Universal Robots PolyScope program: weigh_single_new2.urp

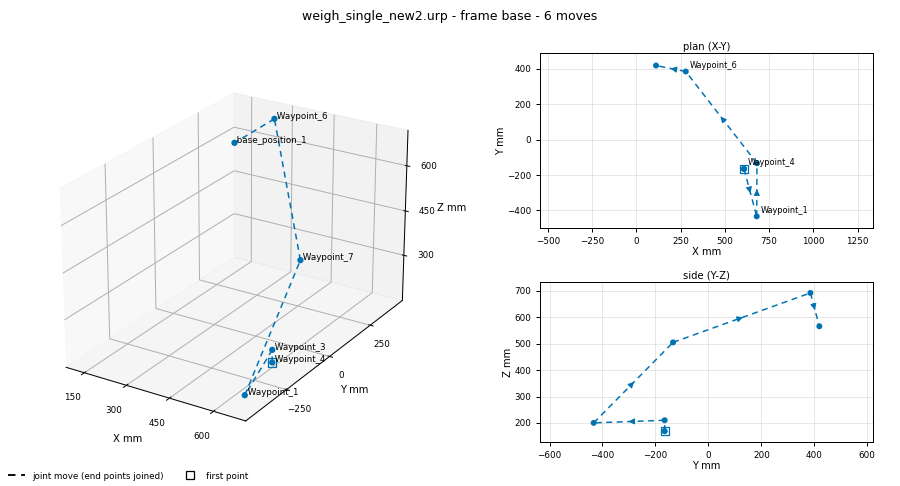
[picture p0: tool path of weigh_single_new2.urp in frame base, 6 of 6 moves have a stored position in this frame; points joined in program order, loops and branches not executed]
Program weigh_single_new2 (installation=default directory=/programs/Nicolas_Arteaga/quality createdIn=5.12.4.1101661 lastSavedIn=5.12.4.1101661 robotSerialNumber=20225502378)
Calibrated DH parameters: a=[0.00022, -0.425328, -0.389701, 0.000059, 0.000065, 0]; d=[0.162608, 0.803456, 9.992211, -10.662202, 0.099702, 0.099559]; alpha=[1.570756, 0.001543, 0.004316, 1.570651, -1.570122, 0]; deltaTheta=[0, 0.002917, 0.116094, -0.119008, 0, -0.000001]
Robot Program (runOnlyOnce=true)
  MoveJ speed 60 deg/s, acceleration 80 deg/s^2 (useActiveTCP=true) feature=Base
    URCap Gripper (Robotiq_Grippers, Robotiq Inc.) dataModel(position=41.96078431372549, force=100.0, speed=100.0, positionInDouble=41.96078431372549, forceInDouble=100.0, speedInDouble=100.0, slaveIds=[9], blocking=true)
    URCap Gripper (Robotiq_Grippers, Robotiq Inc.) dataModel(position=100.0, force=100.0, speed=100.0, positionInDouble=100.0, forceInDouble=100.0, speedInDouble=100.0, slaveIds=[9], blocking=true)
    Waypoint Waypoint_4: TCP in base x=607.939 y=-165.205 z=168.973 mm, rx=1.2164 ry=1.1511 rz=1.1658 rad; joints [132.859, -78.034, 131.663, -55.503, 46.638, 0.907] deg; TCP offset x=0 y=0 z=191.5 mm, rx=0 ry=0 rz=0 rad
    Waypoint Waypoint_3: TCP in base x=607.929 y=-165.259 z=210.32 mm, rx=1.2164 ry=1.151 rz=1.1657 rad; joints [132.864, -83.639, 129.414, -47.669, 46.63, 0.933] deg
    Waypoint Waypoint_1: TCP in base x=679.711 y=-433.377 z=200.411 mm, rx=1.5798 ry=-1.255 rz=2.1333 rad; joints [140.592, -60.998, 101.194, -44.002, 97.228, 120.111] deg
    URCap Gripper (Robotiq_Grippers, Robotiq Inc.) dataModel(position=0.0, force=100.0, speed=100.0, positionInDouble=0.0, forceInDouble=100.0, speedInDouble=100.0, slaveIds=[9], blocking=true)
    Wait Sleep waitTime=1
    Waypoint Waypoint_7: TCP in base x=681.109 y=-133.566 z=504.363 mm, rx=1.51 ry=0.5692 rz=1.7051 rad; joints [148.757, -93.294, 99.441, -18.453, 68.562, 44.126] deg
    URCap Gripper (Robotiq_Grippers, Robotiq Inc.) dataModel(position=100.0, force=100.0, speed=100.0, positionInDouble=100.0, forceInDouble=100.0, speedInDouble=100.0, slaveIds=[9], blocking=true)
    Waypoint Waypoint_6: TCP in base x=278.734 y=385.121 z=691.066 mm, rx=-0.517 ry=1.1123 rz=1.6333 rad; joints [180.614, -126.096, 113.581, -55.011, 31.191, 1.845] deg
    Waypoint base_position_1: TCP in base x=110.839 y=418.881 z=565.194 mm, rx=-1.5602 ry=-0.9892 rz=-1.3623 rad; joints [201.946, -128.864, 99.356, 35.835, 42.385, 90.241] deg
    'Finish Pressure Measurements'
